// TIA Portal V20 export
ORGANIZATION_BLOCK "Startup"   // OB1035, LAD, Startup
TITLE = "Complete Restart"
// stored: AutoNumber false, IsIECCheckEnabled true, Namespace Unit1.Em6, SetENOAutomatically true
   VAR_INPUT
      LostRetentive : Bool;   // True if retentive data are lost
      LostRTC : Bool;   // True if date and time are lost
   END_VAR
BEGIN

REGION Network 1 (SCL): Build the Absolut Reference Designator
   // Set the Absoult Reference Designator in the Config DB
   IF LEN(IN := "Unit1.Em6.Config".em.referenceDesignator.parent) <> 0 THEN
       "Unit1.Em6.Config".em.referenceDesignator.combined := CONCAT_WSTRING(IN1 := "Unit1.Em6.Config".em.referenceDesignator.parent, IN2 := WSTRING#'.', IN3 := "Unit1.Em6.Config".em.referenceDesignator.relative);
   ELSE
       "Unit1.Em6.Config".em.referenceDesignator.combined := "Unit1.Em6.Config".em.referenceDesignator.relative;
   END_IF;
END_REGION

REGION Network 2 (SCL): Assign axes data
   // This is an example how to assign axes to DB_ANY in DB Config. If you have axes, assign them here. The Config.axis[] variables will be handed over to the control modules. That enables a flexible programming.
   // Assign axes
   "Unit1.MotionNodes".PLCToMotion.TechnologyObject.Axis.VisionZ := "Unit1.Em6.Config".axis[1] := "BA010AZCRDR9_VisionAxisZ";

   // cam
   "Unit1.MotionNodes".PLCToMotion.TechnologyObject.Cam.VisionZCam:= "Unit1.Em6.Config".cam[1] := "BA010AZCRDR9_VisionAxisZCamMain";

   // OutputCam
   "Unit1.MotionNodes".PLCToMotion.TechnologyObject.OutputCam.VisionZDownOutputCam := "Unit1.Em6.Config".outputCam[1] := "OutputCam_VisionZDown";

   // HW_SubModule
   "Unit1.Em6.Config".moduleAccessPoint[1] := "BA010AZCRCU2~BA010AZARCU2_X150~BA010AZCRDR9_ModuleAccessPoint";

   // FB Enable
   "Unit1.Em6.HmiInterface".cmVisionUnitAxisZ.commands.enableMasterControl := TRUE;

   // Assign configuration Homing
   "Unit1.Em6.ControlNodes".cmVisionUnitAxisZ.commandConfiguration.homing.mode := "Unit1.Em6.HmiInterface".cmVisionUnitAxisZ.commandConfiguration.homing.mode := 3;
END_REGION

REGION Network 3 (SCL): CM Config
   // Vision UnitAxis Z
   "Unit1.Em6.Config".cmVisionUnitAxisZ.referenceDesignator := WSTRING#'Vision Axis Z';
   "Unit1.Em6.Config".cmVisionUnitAxisZ.disableAlarms := FALSE;
   "Unit1.Em6.Config".cmVisionUnitAxisZ.masterControlPopUp := TRUE;


   // Vision Controller
   "Unit1.Em6.Config".cmVisionController.hwID.cmdResultStatusID := "BA010AZCRIKVC1~Command_and_Result_Status_1";
   "Unit1.Em6.Config".cmVisionController.hwID.trgReadyStatusID := "BA010AZCRIKVC1~Trg_Ready_Status_1";
   "Unit1.Em6.Config".cmVisionController.hwID.trgAckStatusID := "BA010AZCRIKVC1~Trg_Ack_Status_1";
   "Unit1.Em6.Config".cmVisionController.hwID.miscellaneousStatusID := "BA010AZCRIKVC1~Miscellaneous_Status_1";
   "Unit1.Em6.Config".cmVisionController.hwID.assignableStatusID := "BA010AZCRIKVC1~Assignable_Status_1";
   "Unit1.Em6.Config".cmVisionController.hwID.resultData248ByteID_1 := "BA010AZCRIKVC1~Result_Data_248Byte_1";
   "Unit1.Em6.Config".cmVisionController.hwID.resultData248ByteID_2 := "BA010AZCRIKVC1~Result_Data_248Byte_2";
   "Unit1.Em6.Config".cmVisionController.hwID.resultData248ByteID_3 := "BA010AZCRIKVC1~Result_Data_248Byte_3";
   "Unit1.Em6.Config".cmVisionController.hwID.resultData248ByteID_4 := "BA010AZCRIKVC1~Result_Data_248Byte_4";
   "Unit1.Em6.Config".cmVisionController.hwID.resultData248ByteID_5 := "BA010AZCRIKVC1~Result_Data_248Byte_5";
   "Unit1.Em6.Config".cmVisionController.hwID.cmdResultControlID := "BA010AZCRIKVC1~Command_and_Result_Control_1";
   "Unit1.Em6.Config".cmVisionController.hwID.trgControlID := "BA010AZCRIKVC1~Trg_Control_1";
   "Unit1.Em6.Config".cmVisionController.hwID.miscellaneousControlID := "BA010AZCRIKVC1~Miscellaneous_Control_1";
   "Unit1.Em6.Config".cmVisionController.hwID.reservedControlID := "BA010AZCRIKVC1~Reserved_Control_1";
   "Unit1.Em6.Config".cmVisionController.hwID.assignableControlID := "BA010AZCRIKVC1~Assignable_Control_1";
   "Unit1.Em6.Config".cmVisionController.hwID.parameterData248ByteID_1 := "BA010AZCRIKVC1~Parameter_248Byte_1";
   "Unit1.Em6.Config".cmVisionController.hwID.parameterData248ByteID_2 := "BA010AZCRIKVC1~Parameter_248Byte_2";
   "Unit1.Em6.Config".cmVisionController.hwID.parameterData248ByteID_3 := "BA010AZCRIKVC1~Parameter_248Byte_3";
   "Unit1.Em6.Config".cmVisionController.hwID.parameterData248ByteID_4 := "BA010AZCRIKVC1~Parameter_248Byte_4";
   "Unit1.Em6.Config".cmVisionController.hwID.parameterData248ByteID_5 := "BA010AZCRIKVC1~Parameter_248Byte_5";
   "Unit1.Em6.Config".cmVisionController.referenceDesignator := WSTRING#'Vision Controller';
   "Unit1.Em6.Config".cmVisionController.disableAlarms := FALSE;
   "Unit1.Em6.Config".cmVisionController.trigger1Use := TRUE;
   "Unit1.Em6.Config".cmVisionController.trigger2Use := FALSE;
   "Unit1.Em6.Config".cmVisionController.trigger3Use := FALSE;
   "Unit1.Em6.Config".cmVisionController.trigger4Use := FALSE;
   "Unit1.Em6.Config".cmVisionController.triggertime := T#5ms;
   "Unit1.Em6.Config".cmVisionController.cycleTime := T#750ms;


   // QR Reader Fix
   // Config.cmQrReadFix.handshakeGeneralErrorStatusHwId := _."BA020AZCRICAMPN01~Handshake_and_General_Error_Status_,,,";
   // Config.cmQrReadFix.busyStatusHwId := _."BA020AZCRICAMPN01~BUSY_Status_Bits_1";
   // Config.cmQrReadFix.completionStatusHwId := _."BA020AZCRICAMPN01~Completion_Status_Bits_1";
   // Config.cmQrReadFix.errorStatusHwId := _."BA020AZCRICAMPN01~Reserved_1_1";
   // Config.cmQrReadFix.terminalStatusHwId := _."BA020AZCRICAMPN01~Terminal_Status_Bits_1";
   // Config.cmQrReadFix.unstableReadStatusHwId := _."BA020AZCRICAMPN01~Unstable_Read_Status_Bits_1";
   // Config.cmQrReadFix.matchingAndGradeStatusHwId := _."BA020AZCRICAMPN01~Matching_Level_and_Total_Evaluation,,,";
   // Config.cmQrReadFix.operationResultStatusHwId := _."BA020AZCRICAMPN01~Operation_Result_Status_1";
   // Config.cmQrReadFix.readDataHeaderHwId := _."BA020AZCRICAMPN01~Read_Data_128Byte_1";
   // Config.cmQrReadFix.latchErrorClearControlHwId := _."BA020AZCRICAMPN01~Latch_and_Error_Clear_Control_Bits_1";
   // Config.cmQrReadFix.operationInstructionControlHwId := _."BA020AZCRICAMPN01~Operation_instruction_Control_Bits_1";
   // Config.cmQrReadFix.completionClearControlHwId := _."BA020AZCRICAMPN01~Completion_Clear_Control_Bits_1";
   // Config.cmQrReadFix.parameterBankNumberHwId := _."BA020AZCRICAMPN01~Parameter_Bank_Number_1";
   // Config.cmQrReadFix.userDataHwId := _."BA020AZCRICAMPN01~User_Data_128Byte_1";
   "Unit1.Em6.Config".cmQrReader.referenceDesignator := WSTRING#'QR Reader Fix';
   "Unit1.Em6.Config".cmQrReader.triggertime := T#5ms;
   "Unit1.Em6.Config".cmQrReader.cycleTime := T#750ms;


   // QR Reader Handy
   // Config.cmQrReadHandy.Acquisition_Status_HW_ID := _."BA010AZARHS1~Acquisition_Status_1";
   // Config.cmQrReadHandy.Results_Status_HW_ID := _."BA010AZARHS1~Results_Status_1";
   // Config.cmQrReadHandy.Soft_Event_Status_HW_ID := _."BA010AZARHS1~Soft_Event_Control_1";
   // Config.cmQrReadHandy.Result_Data_HW_ID := _."BA010AZARHS1~Result_Data_-_64_bytes_1";
   // Config.cmQrReadHandy.Acquisition_Control_HW_ID := _."BA010AZARHS1~Acquisition_Control_1";
   // Config.cmQrReadHandy.Results_Control_HW_ID := _."BA010AZARHS1~Results_Control_1";
   // Config.cmQrReadHandy.Soft_Event_Control_HW_ID := _."BA010AZARHS1~Soft_Event_Control_1";
   // Config.cmQrReadHandy.User_Data_HW_ID := _."BA010AZARHS1~User_Data_-_64_bytes_1";
   "Unit1.Em6.Config".cmQrReaderHandy.referenceDesignator := WSTRING#'QR Reader Handy';
   "Unit1.Em6.Config".cmQrReaderHandy.triggertime := T#5ms;
   "Unit1.Em6.Config".cmQrReaderHandy.cycleTime := T#10s;


   // Vision Pusher Support
   "Unit1.Em6.Config".cmVisionPusherSupportUpDown.referenceDesignator := WSTRING#'Vision Pusher Support';
   "Unit1.Em6.Config".cmVisionPusherSupportUpDown.monitoringLeavingFeedback := T#0ms;
   "Unit1.Em6.Config".cmVisionPusherSupportUpDown.monitoringReachingFeedback := T#0ms;
   "Unit1.Em6.Config".cmVisionPusherSupportUpDown.monitoringDiscrepancy := T#0ms;
   "Unit1.Em6.Config".cmVisionPusherSupportUpDown.setOutputHomeContinuously := TRUE;
   "Unit1.Em6.Config".cmVisionPusherSupportUpDown.setOutputWorkContinuously := TRUE;
   "Unit1.Em6.Config".cmVisionPusherSupportUpDown.disableHomeCommand := FALSE;
   "Unit1.Em6.Config".cmVisionPusherSupportUpDown.disableFeedbackHomePos := TRUE;
   "Unit1.Em6.Config".cmVisionPusherSupportUpDown.disableFeedbackWorkPos := TRUE;
   "Unit1.Em6.Config".cmVisionPusherSupportUpDown.disableAlarms := TRUE;
   "Unit1.Em6.Config".cmVisionPusherSupportUpDown.resetOutputsOnError := FALSE;
   "Unit1.Em6.Config".cmVisionPusherSupportUpDown.allwaysWaitOnReachingTime := FALSE;


   // Vision Trigger Sensor
   "Unit1.Em6.Config".cmVisionTriggerSensor.referenceDesignator := WSTRING#'DigitalSignal';
   "Unit1.Em6.Config".cmVisionTriggerSensor.onDelay := T#0ms;
   "Unit1.Em6.Config".cmVisionTriggerSensor.offDelay := T#0ms;
   "Unit1.Em6.Config".cmVisionTriggerSensor.default := FALSE;
   "Unit1.Em6.Config".cmVisionTriggerSensor.invertProcessValue := FALSE;
   "Unit1.Em6.Config".cmVisionTriggerSensor.disableAlarms := FALSE;


   // Alarm Count referenceDesignator
   "Unit1.Em6.HmiInterface".visionTriggerSensorNotDetectedCount.referenceDesignator := WSTRING#'Vision Trigger Sensor Not Detected Count';


   // Softcam
   //HmiInterface.VisionUnitAxisZSoftCam.UnitName := WSTRING#'°';
END_REGION
END_ORGANIZATION_BLOCK
